TYPE EL5101_ControlChannel :
STRUCT
	{attribute addProperty Name "Control"}
	Control AT %Q* : EL5101_Control;
	{attribute addProperty Name "Set counter value"}
	SetCounterValue AT %Q* : UINT;
END_STRUCT
END_TYPE

(* stored: Version 1.1.0.1, ProductVersion 3.1.4024.9
   DUT EL5101_ControlChannel: Id {b6d7b352-9606-0aee-367f-b6ab0007318e} *)
